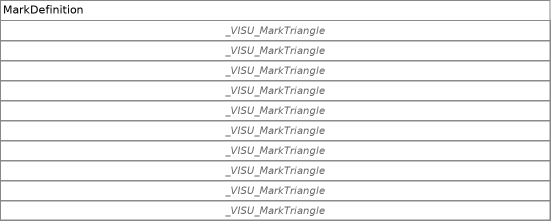
VISUALIZATION _VISU_MarkDefinition  // 551x221
VAR_IN_OUT
	mInst : FB_MarkDefinition;
END_VAR
    Frame (0,20 551x21)
        shows _VISU_MarkTriangle(mInst := mInst.sMarkDef[1])
    Frame (0,40 551x21)
        shows _VISU_MarkTriangle(mInst := mInst.sMarkDef[2])
    Frame (0,60 551x21)
        shows _VISU_MarkTriangle(mInst := mInst.sMarkDef[3])
    Frame (0,120 551x21)
        shows _VISU_MarkTriangle(mInst := mInst.sMarkDef[6])
    Frame (0,80 551x21)
        shows _VISU_MarkTriangle(mInst := mInst.sMarkDef[4])
    Frame (0,100 551x21)
        shows _VISU_MarkTriangle(mInst := mInst.sMarkDef[5])
    Frame (0,140 551x21)
        shows _VISU_MarkTriangle(mInst := mInst.sMarkDef[7])
    Frame (0,200 551x21)
        shows _VISU_MarkTriangle(mInst := mInst.sMarkDef[10])
    Frame (0,160 551x21)
        shows _VISU_MarkTriangle(mInst := mInst.sMarkDef[8])
    Frame (0,180 551x21)
        shows _VISU_MarkTriangle(mInst := mInst.sMarkDef[9])
    Rectangle (0,0 120x20), "MarkDefinition"
END_VISUALIZATION

(* stored: Version 1.1.0.1, ProductVersion 3.1.4024.11
   Visu _VISU_MarkDefinition: Id {8a8bacbe-91d5-4738-bd8e-a2e24cdc1b8d} *)
